// TIA Portal V17 export
// export: Created 2025-03-18T12:31:06.7094667Z, ExportSetting WithDefaults, DisplayName Totally Integrated Automation Portal, DisplayVersion V17 Update 8, DisplayName TIA Portal Openness, DisplayVersion V17 Update 8, DisplayName TIA Portal Version Control Interface, DisplayVersion V17, DisplayName SINAMICS Startdrive Advanced, DisplayVersion V17 SP2, DisplayName SINAMICS Startdrive G110M, G120, G120C, G120D, G120P, G115D, DisplayVersion V17 SP2, DisplayName SINAMICS Startdrive G130, G150, S120, S150, SINAMICS MV, S210, DisplayVersion V17 SP2, DisplayName STEP 7 Professional, DisplayVersion V17 Update 8, DisplayName SINUMERIK ONE STEP 7 Toolbox, DisplayVersion V17 Update 12, DisplayName SINUMERIK 840D sl STEP 7 Toolbox, DisplayVersion V17 Update 12, DisplayName STEP 7 Safety, DisplayVersion V17 Update 6, DisplayName WinCC Advanced, DisplayVersion V17 Update 8
FUNCTION "FC1312_HOME_UNIT_03_STATION_0" : Void   // FC1312, LAD
{ S7_Optimized_Access := 'FALSE' }
AUTHOR : ETXETAR
VERSION : 1.0
// stored: AutoNumber false, IsIECCheckEnabled false, SetENOAutomatically false, UDAEnableTagReadback false
   VAR_TEMP
      UNIT_03_LOCAL_E_RETURNS : Bool;   // UNIT 03 LOCAL E RETURNS
      UNIT_03_MACHINE_E_RETURNS : Bool;   // UNIT 03 MACHINE E RETURNS
   END_VAR
   VAR CONSTANT
      FC_NUMBER : DInt := 1312;
   END_VAR
   VAR_TEMP   // added for the SCL form of the ladder/FBD networks
      _w1 : Bool;
   END_VAR
BEGIN

REGION Network 1: GENERAL CONDITIONS
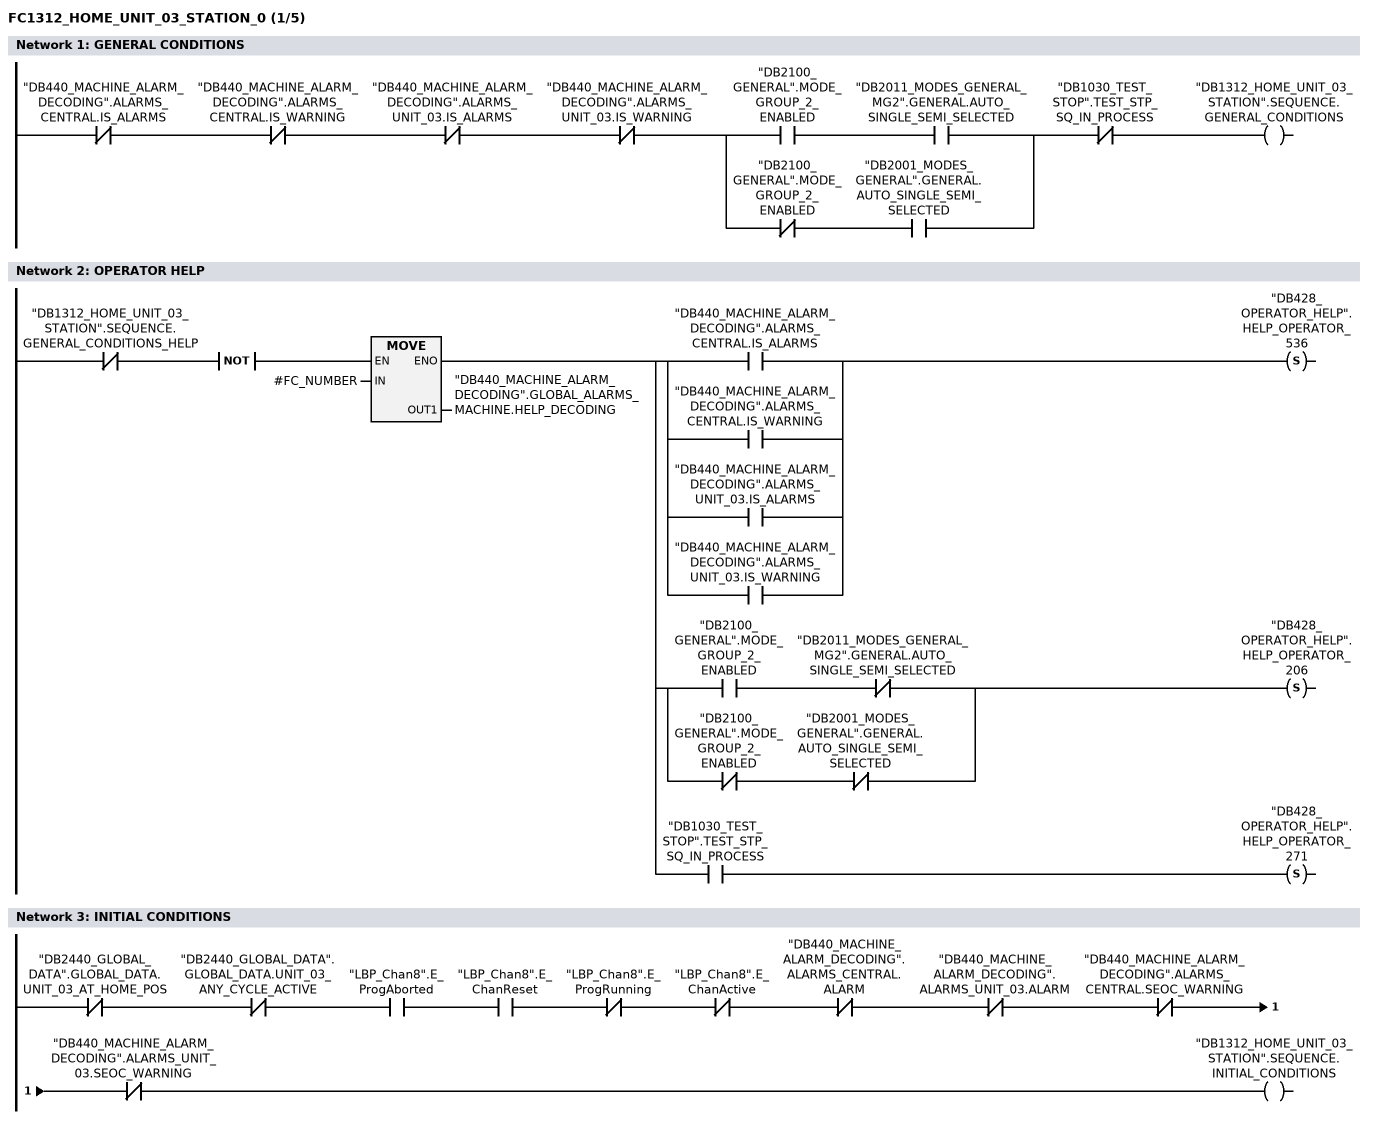
   RUNG wire#powerrail
      I_Contact( "DB440_MACHINE_ALARM_DECODING".ALARMS_CENTRAL.IS_ALARMS )
      I_Contact( "DB440_MACHINE_ALARM_DECODING".ALARMS_CENTRAL.IS_WARNING )
      I_Contact( "DB440_MACHINE_ALARM_DECODING".ALARMS_UNIT_03.IS_ALARMS )
      I_Contact( "DB440_MACHINE_ALARM_DECODING".ALARMS_UNIT_03.IS_WARNING )
      wire#w1
      Contact( "DB2100_GENERAL".MODE_GROUP_2_ENABLED )
      Contact( "DB2011_MODES_GENERAL_MG2".GENERAL.AUTO_SINGLE_SEMI_SELECTED )
      wire#w2
      I_Contact( "DB1030_TEST_STOP".TEST_STP_SQ_IN_PROCESS )
      Coil( "DB1312_HOME_UNIT_03_STATION".SEQUENCE.GENERAL_CONDITIONS )
   END_RUNG
   RUNG wire#w1
      I_Contact( "DB2100_GENERAL".MODE_GROUP_2_ENABLED )
      Contact( "DB2001_MODES_GENERAL".GENERAL.AUTO_SINGLE_SEMI_SELECTED )
   END_RUNG wire#w2
   // the same network as SCL:
   "DB1312_HOME_UNIT_03_STATION".SEQUENCE.GENERAL_CONDITIONS := NOT "DB440_MACHINE_ALARM_DECODING".ALARMS_CENTRAL.IS_ALARMS AND NOT "DB440_MACHINE_ALARM_DECODING".ALARMS_CENTRAL.IS_WARNING AND NOT "DB440_MACHINE_ALARM_DECODING".ALARMS_UNIT_03.IS_ALARMS AND NOT "DB440_MACHINE_ALARM_DECODING".ALARMS_UNIT_03.IS_WARNING AND (("DB2100_GENERAL".MODE_GROUP_2_ENABLED AND "DB2011_MODES_GENERAL_MG2".GENERAL.AUTO_SINGLE_SEMI_SELECTED) OR (NOT "DB2100_GENERAL".MODE_GROUP_2_ENABLED AND "DB2001_MODES_GENERAL".GENERAL.AUTO_SINGLE_SEMI_SELECTED)) AND NOT "DB1030_TEST_STOP".TEST_STP_SQ_IN_PROCESS;
END_REGION

REGION Network 2: OPERATOR HELP
   RUNG wire#powerrail
      I_Contact( "DB1312_HOME_UNIT_03_STATION".SEQUENCE.GENERAL_CONDITIONS_HELP )
      Not()
      { S7_GenerateENO := "TRUE" } Move(in := #FC_NUMBER, out1 => "DB440_MACHINE_ALARM_DECODING".GLOBAL_ALARMS_MACHINE.HELP_DECODING)
      wire#w1
      Contact( "DB440_MACHINE_ALARM_DECODING".ALARMS_CENTRAL.IS_ALARMS )
      wire#w2
      S_Coil( "DB428_OPERATOR_HELP".HELP_OPERATOR_536 )
   END_RUNG
   RUNG wire#w1
      Contact( "DB440_MACHINE_ALARM_DECODING".ALARMS_CENTRAL.IS_WARNING )
   END_RUNG wire#w2
   RUNG wire#w1
      Contact( "DB440_MACHINE_ALARM_DECODING".ALARMS_UNIT_03.IS_ALARMS )
   END_RUNG wire#w2
   RUNG wire#w1
      Contact( "DB440_MACHINE_ALARM_DECODING".ALARMS_UNIT_03.IS_WARNING )
   END_RUNG wire#w2
   RUNG wire#w1
      Contact( "DB2100_GENERAL".MODE_GROUP_2_ENABLED )
      I_Contact( "DB2011_MODES_GENERAL_MG2".GENERAL.AUTO_SINGLE_SEMI_SELECTED )
      wire#w3
      S_Coil( "DB428_OPERATOR_HELP".HELP_OPERATOR_206 )
   END_RUNG
   RUNG wire#w1
      I_Contact( "DB2100_GENERAL".MODE_GROUP_2_ENABLED )
      I_Contact( "DB2001_MODES_GENERAL".GENERAL.AUTO_SINGLE_SEMI_SELECTED )
   END_RUNG wire#w3
   RUNG wire#w1
      Contact( "DB1030_TEST_STOP".TEST_STP_SQ_IN_PROCESS )
      S_Coil( "DB428_OPERATOR_HELP".HELP_OPERATOR_271 )
   END_RUNG
   // the same network as SCL:
   // ENO of a box is taken as its EN; it also drops when the box reports an error
   #_w1 := NOT (NOT "DB1312_HOME_UNIT_03_STATION".SEQUENCE.GENERAL_CONDITIONS_HELP);
   IF #_w1 THEN "DB440_MACHINE_ALARM_DECODING".GLOBAL_ALARMS_MACHINE.HELP_DECODING := #FC_NUMBER; END_IF;
   IF #_w1 AND ("DB440_MACHINE_ALARM_DECODING".ALARMS_CENTRAL.IS_ALARMS OR "DB440_MACHINE_ALARM_DECODING".ALARMS_CENTRAL.IS_WARNING OR "DB440_MACHINE_ALARM_DECODING".ALARMS_UNIT_03.IS_ALARMS OR "DB440_MACHINE_ALARM_DECODING".ALARMS_UNIT_03.IS_WARNING) THEN
       "DB428_OPERATOR_HELP".HELP_OPERATOR_536 := TRUE;
   END_IF;
   IF #_w1 AND (("DB2100_GENERAL".MODE_GROUP_2_ENABLED AND NOT "DB2011_MODES_GENERAL_MG2".GENERAL.AUTO_SINGLE_SEMI_SELECTED) OR (NOT "DB2100_GENERAL".MODE_GROUP_2_ENABLED AND NOT "DB2001_MODES_GENERAL".GENERAL.AUTO_SINGLE_SEMI_SELECTED)) THEN
       "DB428_OPERATOR_HELP".HELP_OPERATOR_206 := TRUE;
   END_IF;
   IF #_w1 AND "DB1030_TEST_STOP".TEST_STP_SQ_IN_PROCESS THEN
       "DB428_OPERATOR_HELP".HELP_OPERATOR_271 := TRUE;
   END_IF;
END_REGION

REGION Network 3: INITIAL CONDITIONS
   RUNG wire#powerrail
      I_Contact( "DB2440_GLOBAL_DATA".GLOBAL_DATA.UNIT_03_AT_HOME_POS )
      I_Contact( "DB2440_GLOBAL_DATA".GLOBAL_DATA.UNIT_03_ANY_CYCLE_ACTIVE )
      Contact( "LBP_Chan8".E_ProgAborted )
      Contact( "LBP_Chan8".E_ChanReset )
      I_Contact( "LBP_Chan8".E_ProgRunning )
      I_Contact( "LBP_Chan8".E_ChanActive )
      I_Contact( "DB440_MACHINE_ALARM_DECODING".ALARMS_CENTRAL.ALARM )
      I_Contact( "DB440_MACHINE_ALARM_DECODING".ALARMS_UNIT_03.ALARM )
      I_Contact( "DB440_MACHINE_ALARM_DECODING".ALARMS_CENTRAL.SEOC_WARNING )
      I_Contact( "DB440_MACHINE_ALARM_DECODING".ALARMS_UNIT_03.SEOC_WARNING )
      Coil( "DB1312_HOME_UNIT_03_STATION".SEQUENCE.INITIAL_CONDITIONS )
   END_RUNG
   // the same network as SCL:
   "DB1312_HOME_UNIT_03_STATION".SEQUENCE.INITIAL_CONDITIONS := NOT "DB2440_GLOBAL_DATA".GLOBAL_DATA.UNIT_03_AT_HOME_POS AND NOT "DB2440_GLOBAL_DATA".GLOBAL_DATA.UNIT_03_ANY_CYCLE_ACTIVE AND "LBP_Chan8".E_ProgAborted AND "LBP_Chan8".E_ChanReset AND NOT "LBP_Chan8".E_ProgRunning AND NOT "LBP_Chan8".E_ChanActive AND NOT "DB440_MACHINE_ALARM_DECODING".ALARMS_CENTRAL.ALARM AND NOT "DB440_MACHINE_ALARM_DECODING".ALARMS_UNIT_03.ALARM AND NOT "DB440_MACHINE_ALARM_DECODING".ALARMS_CENTRAL.SEOC_WARNING AND NOT "DB440_MACHINE_ALARM_DECODING".ALARMS_UNIT_03.SEOC_WARNING;
END_REGION

REGION Network 4: OPERATOR HELP
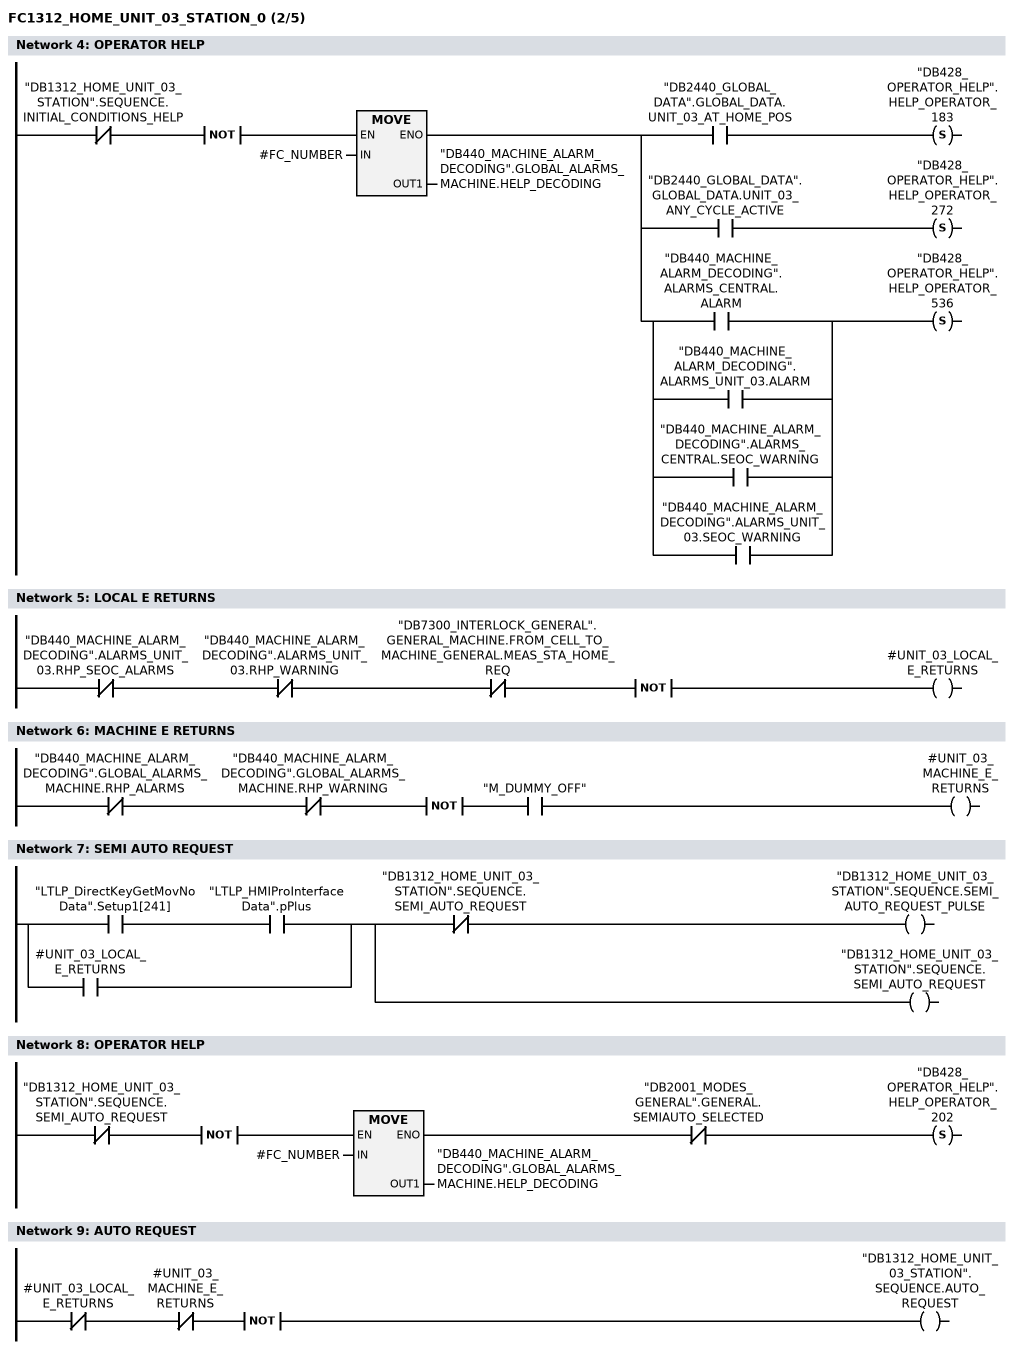
   RUNG wire#powerrail
      I_Contact( "DB1312_HOME_UNIT_03_STATION".SEQUENCE.INITIAL_CONDITIONS_HELP )
      Not()
      { S7_GenerateENO := "TRUE" } Move(in := #FC_NUMBER, out1 => "DB440_MACHINE_ALARM_DECODING".GLOBAL_ALARMS_MACHINE.HELP_DECODING)
      wire#w1
      Contact( "DB2440_GLOBAL_DATA".GLOBAL_DATA.UNIT_03_AT_HOME_POS )
      S_Coil( "DB428_OPERATOR_HELP".HELP_OPERATOR_183 )
   END_RUNG
   RUNG wire#w1
      Contact( "DB2440_GLOBAL_DATA".GLOBAL_DATA.UNIT_03_ANY_CYCLE_ACTIVE )
      S_Coil( "DB428_OPERATOR_HELP".HELP_OPERATOR_272 )
   END_RUNG
   RUNG wire#w1
      Contact( "DB440_MACHINE_ALARM_DECODING".ALARMS_CENTRAL.ALARM )
      wire#w2
      S_Coil( "DB428_OPERATOR_HELP".HELP_OPERATOR_536 )
   END_RUNG
   RUNG wire#w1
      Contact( "DB440_MACHINE_ALARM_DECODING".ALARMS_UNIT_03.ALARM )
   END_RUNG wire#w2
   RUNG wire#w1
      Contact( "DB440_MACHINE_ALARM_DECODING".ALARMS_CENTRAL.SEOC_WARNING )
   END_RUNG wire#w2
   RUNG wire#w1
      Contact( "DB440_MACHINE_ALARM_DECODING".ALARMS_UNIT_03.SEOC_WARNING )
   END_RUNG wire#w2
   // the same network as SCL:
   // ENO of a box is taken as its EN; it also drops when the box reports an error
   #_w1 := NOT (NOT "DB1312_HOME_UNIT_03_STATION".SEQUENCE.INITIAL_CONDITIONS_HELP);
   IF #_w1 THEN "DB440_MACHINE_ALARM_DECODING".GLOBAL_ALARMS_MACHINE.HELP_DECODING := #FC_NUMBER; END_IF;
   IF #_w1 AND "DB2440_GLOBAL_DATA".GLOBAL_DATA.UNIT_03_AT_HOME_POS THEN
       "DB428_OPERATOR_HELP".HELP_OPERATOR_183 := TRUE;
   END_IF;
   IF #_w1 AND "DB2440_GLOBAL_DATA".GLOBAL_DATA.UNIT_03_ANY_CYCLE_ACTIVE THEN
       "DB428_OPERATOR_HELP".HELP_OPERATOR_272 := TRUE;
   END_IF;
   IF #_w1 AND ("DB440_MACHINE_ALARM_DECODING".ALARMS_CENTRAL.ALARM OR "DB440_MACHINE_ALARM_DECODING".ALARMS_UNIT_03.ALARM OR "DB440_MACHINE_ALARM_DECODING".ALARMS_CENTRAL.SEOC_WARNING OR "DB440_MACHINE_ALARM_DECODING".ALARMS_UNIT_03.SEOC_WARNING) THEN
       "DB428_OPERATOR_HELP".HELP_OPERATOR_536 := TRUE;
   END_IF;
END_REGION

REGION Network 5: LOCAL E RETURNS
   RUNG wire#powerrail
      I_Contact( "DB440_MACHINE_ALARM_DECODING".ALARMS_UNIT_03.RHP_SEOC_ALARMS )
      I_Contact( "DB440_MACHINE_ALARM_DECODING".ALARMS_UNIT_03.RHP_WARNING )
      I_Contact( "DB7300_INTERLOCK_GENERAL".GENERAL_MACHINE.FROM_CELL_TO_MACHINE_GENERAL.MEAS_STA_HOME_REQ )
      Not()
      Coil( #UNIT_03_LOCAL_E_RETURNS )
   END_RUNG
   // the same network as SCL:
   #UNIT_03_LOCAL_E_RETURNS := NOT (NOT "DB440_MACHINE_ALARM_DECODING".ALARMS_UNIT_03.RHP_SEOC_ALARMS AND NOT "DB440_MACHINE_ALARM_DECODING".ALARMS_UNIT_03.RHP_WARNING AND NOT "DB7300_INTERLOCK_GENERAL".GENERAL_MACHINE.FROM_CELL_TO_MACHINE_GENERAL.MEAS_STA_HOME_REQ);
END_REGION

REGION Network 6: MACHINE E RETURNS
   RUNG wire#powerrail
      I_Contact( "DB440_MACHINE_ALARM_DECODING".GLOBAL_ALARMS_MACHINE.RHP_ALARMS )
      I_Contact( "DB440_MACHINE_ALARM_DECODING".GLOBAL_ALARMS_MACHINE.RHP_WARNING )
      Not()
      Contact( "M_DUMMY_OFF" )
      Coil( #UNIT_03_MACHINE_E_RETURNS )
   END_RUNG
   // the same network as SCL:
   #UNIT_03_MACHINE_E_RETURNS := NOT (NOT "DB440_MACHINE_ALARM_DECODING".GLOBAL_ALARMS_MACHINE.RHP_ALARMS AND NOT "DB440_MACHINE_ALARM_DECODING".GLOBAL_ALARMS_MACHINE.RHP_WARNING) AND "M_DUMMY_OFF";
END_REGION

REGION Network 7: SEMI AUTO REQUEST
   RUNG wire#powerrail
      Contact( "LTLP_DirectKeyGetMovNoData".Setup1[241] )
      Contact( "LTLP_HMIProInterfaceData".pPlus )
      wire#w1
      I_Contact( "DB1312_HOME_UNIT_03_STATION".SEQUENCE.SEMI_AUTO_REQUEST )
      Coil( "DB1312_HOME_UNIT_03_STATION".SEQUENCE.SEMI_AUTO_REQUEST_PULSE )
   END_RUNG
   RUNG wire#powerrail
      Contact( #UNIT_03_LOCAL_E_RETURNS )
   END_RUNG wire#w1
   RUNG wire#w1
      Coil( "DB1312_HOME_UNIT_03_STATION".SEQUENCE.SEMI_AUTO_REQUEST )
   END_RUNG
   // the same network as SCL:
   #_w1 := ("LTLP_DirectKeyGetMovNoData".Setup1[241] AND "LTLP_HMIProInterfaceData".pPlus) OR #UNIT_03_LOCAL_E_RETURNS;
   "DB1312_HOME_UNIT_03_STATION".SEQUENCE.SEMI_AUTO_REQUEST_PULSE := #_w1 AND NOT "DB1312_HOME_UNIT_03_STATION".SEQUENCE.SEMI_AUTO_REQUEST;
   "DB1312_HOME_UNIT_03_STATION".SEQUENCE.SEMI_AUTO_REQUEST := #_w1;
END_REGION

REGION Network 8: OPERATOR HELP
   RUNG wire#powerrail
      I_Contact( "DB1312_HOME_UNIT_03_STATION".SEQUENCE.SEMI_AUTO_REQUEST )
      Not()
      { S7_GenerateENO := "TRUE" } Move(in := #FC_NUMBER, out1 => "DB440_MACHINE_ALARM_DECODING".GLOBAL_ALARMS_MACHINE.HELP_DECODING)
      I_Contact( "DB2001_MODES_GENERAL".GENERAL.SEMIAUTO_SELECTED )
      S_Coil( "DB428_OPERATOR_HELP".HELP_OPERATOR_202 )
   END_RUNG
   // the same network as SCL:
   // ENO of a box is taken as its EN; it also drops when the box reports an error
   #_w1 := NOT (NOT "DB1312_HOME_UNIT_03_STATION".SEQUENCE.SEMI_AUTO_REQUEST);
   IF #_w1 THEN "DB440_MACHINE_ALARM_DECODING".GLOBAL_ALARMS_MACHINE.HELP_DECODING := #FC_NUMBER; END_IF;
   IF #_w1 AND NOT "DB2001_MODES_GENERAL".GENERAL.SEMIAUTO_SELECTED THEN
       "DB428_OPERATOR_HELP".HELP_OPERATOR_202 := TRUE;
   END_IF;
END_REGION

REGION Network 9: AUTO REQUEST
   RUNG wire#powerrail
      I_Contact( #UNIT_03_LOCAL_E_RETURNS )
      I_Contact( #UNIT_03_MACHINE_E_RETURNS )
      Not()
      Coil( "DB1312_HOME_UNIT_03_STATION".SEQUENCE.AUTO_REQUEST )
   END_RUNG
   // the same network as SCL:
   "DB1312_HOME_UNIT_03_STATION".SEQUENCE.AUTO_REQUEST := NOT (NOT #UNIT_03_LOCAL_E_RETURNS AND NOT #UNIT_03_MACHINE_E_RETURNS);
END_REGION

REGION Network 10: REQUEST
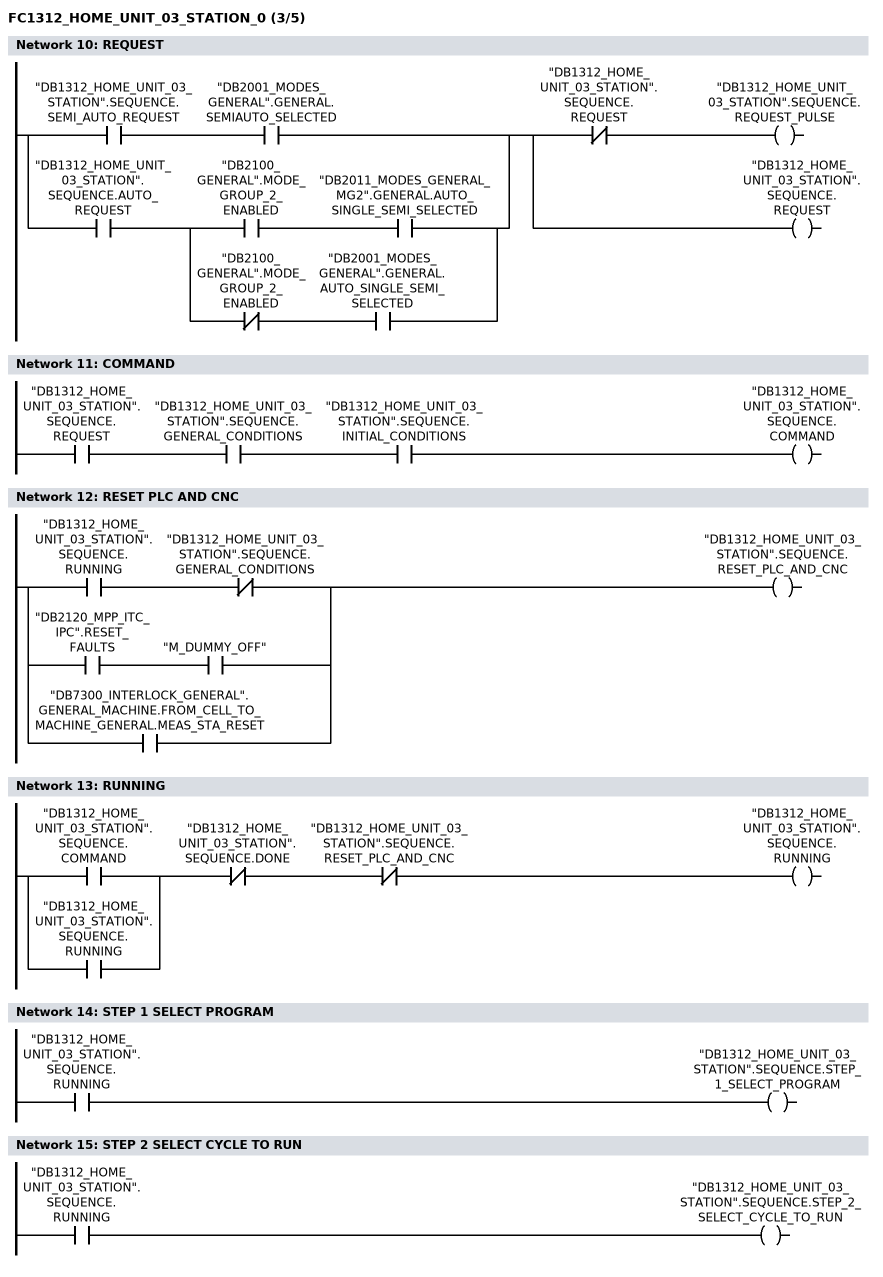
   RUNG wire#powerrail
      Contact( "DB1312_HOME_UNIT_03_STATION".SEQUENCE.SEMI_AUTO_REQUEST )
      Contact( "DB2001_MODES_GENERAL".GENERAL.SEMIAUTO_SELECTED )
      wire#w1
      I_Contact( "DB1312_HOME_UNIT_03_STATION".SEQUENCE.REQUEST )
      Coil( "DB1312_HOME_UNIT_03_STATION".SEQUENCE.REQUEST_PULSE )
   END_RUNG
   RUNG wire#powerrail
      Contact( "DB1312_HOME_UNIT_03_STATION".SEQUENCE.AUTO_REQUEST )
      wire#w2
      Contact( "DB2100_GENERAL".MODE_GROUP_2_ENABLED )
      Contact( "DB2011_MODES_GENERAL_MG2".GENERAL.AUTO_SINGLE_SEMI_SELECTED )
   END_RUNG wire#w1
   RUNG wire#w2
      I_Contact( "DB2100_GENERAL".MODE_GROUP_2_ENABLED )
      Contact( "DB2001_MODES_GENERAL".GENERAL.AUTO_SINGLE_SEMI_SELECTED )
   END_RUNG wire#w1
   RUNG wire#w1
      Coil( "DB1312_HOME_UNIT_03_STATION".SEQUENCE.REQUEST )
   END_RUNG
   // the same network as SCL:
   #_w1 := ("DB1312_HOME_UNIT_03_STATION".SEQUENCE.SEMI_AUTO_REQUEST AND "DB2001_MODES_GENERAL".GENERAL.SEMIAUTO_SELECTED) OR ("DB1312_HOME_UNIT_03_STATION".SEQUENCE.AUTO_REQUEST AND (("DB2100_GENERAL".MODE_GROUP_2_ENABLED AND "DB2011_MODES_GENERAL_MG2".GENERAL.AUTO_SINGLE_SEMI_SELECTED) OR (NOT "DB2100_GENERAL".MODE_GROUP_2_ENABLED AND "DB2001_MODES_GENERAL".GENERAL.AUTO_SINGLE_SEMI_SELECTED)));
   "DB1312_HOME_UNIT_03_STATION".SEQUENCE.REQUEST_PULSE := #_w1 AND NOT "DB1312_HOME_UNIT_03_STATION".SEQUENCE.REQUEST;
   "DB1312_HOME_UNIT_03_STATION".SEQUENCE.REQUEST := #_w1;
END_REGION

REGION Network 11: COMMAND
   RUNG wire#powerrail
      Contact( "DB1312_HOME_UNIT_03_STATION".SEQUENCE.REQUEST )
      Contact( "DB1312_HOME_UNIT_03_STATION".SEQUENCE.GENERAL_CONDITIONS )
      Contact( "DB1312_HOME_UNIT_03_STATION".SEQUENCE.INITIAL_CONDITIONS )
      Coil( "DB1312_HOME_UNIT_03_STATION".SEQUENCE.COMMAND )
   END_RUNG
   // the same network as SCL:
   "DB1312_HOME_UNIT_03_STATION".SEQUENCE.COMMAND := "DB1312_HOME_UNIT_03_STATION".SEQUENCE.REQUEST AND "DB1312_HOME_UNIT_03_STATION".SEQUENCE.GENERAL_CONDITIONS AND "DB1312_HOME_UNIT_03_STATION".SEQUENCE.INITIAL_CONDITIONS;
END_REGION

REGION Network 12: RESET PLC AND CNC
   RUNG wire#powerrail
      Contact( "DB1312_HOME_UNIT_03_STATION".SEQUENCE.RUNNING )
      I_Contact( "DB1312_HOME_UNIT_03_STATION".SEQUENCE.GENERAL_CONDITIONS )
      wire#w1
      Coil( "DB1312_HOME_UNIT_03_STATION".SEQUENCE.RESET_PLC_AND_CNC )
   END_RUNG
   RUNG wire#powerrail
      Contact( "DB2120_MPP_ITC_IPC".RESET_FAULTS )
      Contact( "M_DUMMY_OFF" )
   END_RUNG wire#w1
   RUNG wire#powerrail
      Contact( "DB7300_INTERLOCK_GENERAL".GENERAL_MACHINE.FROM_CELL_TO_MACHINE_GENERAL.MEAS_STA_RESET )
   END_RUNG wire#w1
   // the same network as SCL:
   "DB1312_HOME_UNIT_03_STATION".SEQUENCE.RESET_PLC_AND_CNC := ("DB1312_HOME_UNIT_03_STATION".SEQUENCE.RUNNING AND NOT "DB1312_HOME_UNIT_03_STATION".SEQUENCE.GENERAL_CONDITIONS) OR ("DB2120_MPP_ITC_IPC".RESET_FAULTS AND "M_DUMMY_OFF") OR "DB7300_INTERLOCK_GENERAL".GENERAL_MACHINE.FROM_CELL_TO_MACHINE_GENERAL.MEAS_STA_RESET;
END_REGION

REGION Network 13: RUNNING
   RUNG wire#powerrail
      Contact( "DB1312_HOME_UNIT_03_STATION".SEQUENCE.COMMAND )
      wire#w1
      I_Contact( "DB1312_HOME_UNIT_03_STATION".SEQUENCE.DONE )
      I_Contact( "DB1312_HOME_UNIT_03_STATION".SEQUENCE.RESET_PLC_AND_CNC )
      Coil( "DB1312_HOME_UNIT_03_STATION".SEQUENCE.RUNNING )
   END_RUNG
   RUNG wire#powerrail
      Contact( "DB1312_HOME_UNIT_03_STATION".SEQUENCE.RUNNING )
   END_RUNG wire#w1
   // the same network as SCL:
   "DB1312_HOME_UNIT_03_STATION".SEQUENCE.RUNNING := ("DB1312_HOME_UNIT_03_STATION".SEQUENCE.COMMAND OR "DB1312_HOME_UNIT_03_STATION".SEQUENCE.RUNNING) AND NOT "DB1312_HOME_UNIT_03_STATION".SEQUENCE.DONE AND NOT "DB1312_HOME_UNIT_03_STATION".SEQUENCE.RESET_PLC_AND_CNC;
END_REGION

REGION Network 14: STEP 1 SELECT PROGRAM
   RUNG wire#powerrail
      Contact( "DB1312_HOME_UNIT_03_STATION".SEQUENCE.RUNNING )
      Coil( "DB1312_HOME_UNIT_03_STATION".SEQUENCE.STEP_1_SELECT_PROGRAM )
   END_RUNG
   // the same network as SCL:
   "DB1312_HOME_UNIT_03_STATION".SEQUENCE.STEP_1_SELECT_PROGRAM := "DB1312_HOME_UNIT_03_STATION".SEQUENCE.RUNNING;
END_REGION

REGION Network 15: STEP 2 SELECT CYCLE TO RUN
   RUNG wire#powerrail
      Contact( "DB1312_HOME_UNIT_03_STATION".SEQUENCE.RUNNING )
      Coil( "DB1312_HOME_UNIT_03_STATION".SEQUENCE.STEP_2_SELECT_CYCLE_TO_RUN )
   END_RUNG
   // the same network as SCL:
   "DB1312_HOME_UNIT_03_STATION".SEQUENCE.STEP_2_SELECT_CYCLE_TO_RUN := "DB1312_HOME_UNIT_03_STATION".SEQUENCE.RUNNING;
END_REGION

REGION Network 16: STEP 3 RUN CNC PROGRAM
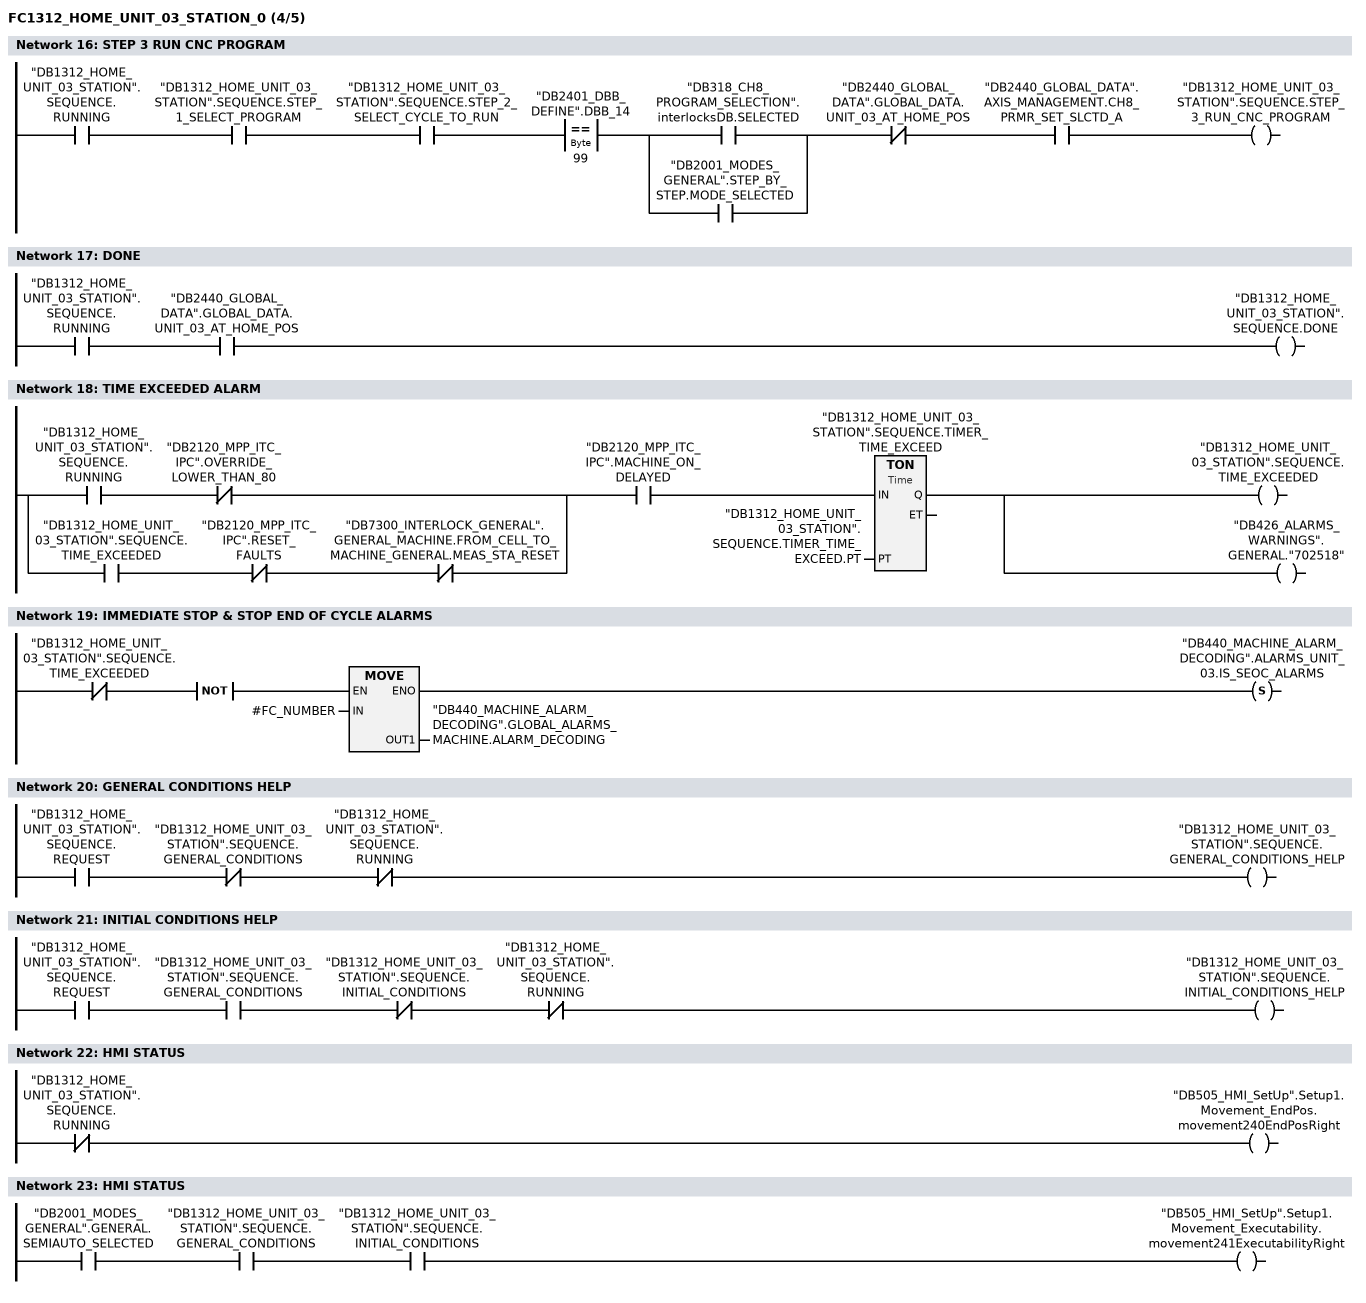
   RUNG wire#powerrail
      Contact( "DB1312_HOME_UNIT_03_STATION".SEQUENCE.RUNNING )
      Contact( "DB1312_HOME_UNIT_03_STATION".SEQUENCE.STEP_1_SELECT_PROGRAM )
      Contact( "DB1312_HOME_UNIT_03_STATION".SEQUENCE.STEP_2_SELECT_CYCLE_TO_RUN )
      { S7_Templates := "SrcType := Byte" } EQ_Contact(in1 := "DB2401_DBB_DEFINE".DBB_14, in2 := 99)
      wire#w1
      Contact( "DB318_CH8_PROGRAM_SELECTION".interlocksDB.SELECTED )
      wire#w2
      I_Contact( "DB2440_GLOBAL_DATA".GLOBAL_DATA.UNIT_03_AT_HOME_POS )
      Contact( "DB2440_GLOBAL_DATA".AXIS_MANAGEMENT.CH8_PRMR_SET_SLCTD_A )
      Coil( "DB1312_HOME_UNIT_03_STATION".SEQUENCE.STEP_3_RUN_CNC_PROGRAM )
   END_RUNG
   RUNG wire#w1
      Contact( "DB2001_MODES_GENERAL".STEP_BY_STEP.MODE_SELECTED )
   END_RUNG wire#w2
   // the same network as SCL:
   "DB1312_HOME_UNIT_03_STATION".SEQUENCE.STEP_3_RUN_CNC_PROGRAM := "DB1312_HOME_UNIT_03_STATION".SEQUENCE.RUNNING AND "DB1312_HOME_UNIT_03_STATION".SEQUENCE.STEP_1_SELECT_PROGRAM AND "DB1312_HOME_UNIT_03_STATION".SEQUENCE.STEP_2_SELECT_CYCLE_TO_RUN AND ("DB2401_DBB_DEFINE".DBB_14 = 99) AND ("DB318_CH8_PROGRAM_SELECTION".interlocksDB.SELECTED OR "DB2001_MODES_GENERAL".STEP_BY_STEP.MODE_SELECTED) AND NOT "DB2440_GLOBAL_DATA".GLOBAL_DATA.UNIT_03_AT_HOME_POS AND "DB2440_GLOBAL_DATA".AXIS_MANAGEMENT.CH8_PRMR_SET_SLCTD_A;
END_REGION

REGION Network 17: DONE
   RUNG wire#powerrail
      Contact( "DB1312_HOME_UNIT_03_STATION".SEQUENCE.RUNNING )
      Contact( "DB2440_GLOBAL_DATA".GLOBAL_DATA.UNIT_03_AT_HOME_POS )
      Coil( "DB1312_HOME_UNIT_03_STATION".SEQUENCE.DONE )
   END_RUNG
   // the same network as SCL:
   "DB1312_HOME_UNIT_03_STATION".SEQUENCE.DONE := "DB1312_HOME_UNIT_03_STATION".SEQUENCE.RUNNING AND "DB2440_GLOBAL_DATA".GLOBAL_DATA.UNIT_03_AT_HOME_POS;
END_REGION

REGION Network 18: TIME EXCEEDED ALARM
   RUNG wire#powerrail
      Contact( "DB1312_HOME_UNIT_03_STATION".SEQUENCE.RUNNING )
      I_Contact( "DB2120_MPP_ITC_IPC".OVERRIDE_LOWER_THAN_80 )
      wire#w1
      Contact( "DB2120_MPP_ITC_IPC".MACHINE_ON_DELAYED )
      { S7_Templates := "time_type := Time" } "DB1312_HOME_UNIT_03_STATION".SEQUENCE.TIMER_TIME_EXCEED.TON(pt := "DB1312_HOME_UNIT_03_STATION".SEQUENCE.TIMER_TIME_EXCEED.PT, et =>)
      wire#w2
      Coil( "DB1312_HOME_UNIT_03_STATION".SEQUENCE.TIME_EXCEEDED )
   END_RUNG
   RUNG wire#powerrail
      Contact( "DB1312_HOME_UNIT_03_STATION".SEQUENCE.TIME_EXCEEDED )
      I_Contact( "DB2120_MPP_ITC_IPC".RESET_FAULTS )
      I_Contact( "DB7300_INTERLOCK_GENERAL".GENERAL_MACHINE.FROM_CELL_TO_MACHINE_GENERAL.MEAS_STA_RESET )
   END_RUNG wire#w1
   RUNG wire#w2
      Coil( "DB426_ALARMS_WARNINGS".GENERAL."702518" )
   END_RUNG
   // the same network as SCL:
   "DB1312_HOME_UNIT_03_STATION".SEQUENCE.TIMER_TIME_EXCEED.TON(IN := (("DB1312_HOME_UNIT_03_STATION".SEQUENCE.RUNNING AND NOT "DB2120_MPP_ITC_IPC".OVERRIDE_LOWER_THAN_80) OR ("DB1312_HOME_UNIT_03_STATION".SEQUENCE.TIME_EXCEEDED AND NOT "DB2120_MPP_ITC_IPC".RESET_FAULTS AND NOT "DB7300_INTERLOCK_GENERAL".GENERAL_MACHINE.FROM_CELL_TO_MACHINE_GENERAL.MEAS_STA_RESET)) AND "DB2120_MPP_ITC_IPC".MACHINE_ON_DELAYED,
                           PT := "DB1312_HOME_UNIT_03_STATION".SEQUENCE.TIMER_TIME_EXCEED.PT);
   "DB1312_HOME_UNIT_03_STATION".SEQUENCE.TIME_EXCEEDED := "DB1312_HOME_UNIT_03_STATION".SEQUENCE.TIMER_TIME_EXCEED.Q;
   "DB426_ALARMS_WARNINGS".GENERAL."702518" := "DB1312_HOME_UNIT_03_STATION".SEQUENCE.TIMER_TIME_EXCEED.Q;
END_REGION

REGION Network 19: IMMEDIATE STOP & STOP END OF CYCLE ALARMS
   RUNG wire#powerrail
      I_Contact( "DB1312_HOME_UNIT_03_STATION".SEQUENCE.TIME_EXCEEDED )
      Not()
      { S7_GenerateENO := "TRUE" } Move(in := #FC_NUMBER, out1 => "DB440_MACHINE_ALARM_DECODING".GLOBAL_ALARMS_MACHINE.ALARM_DECODING)
      S_Coil( "DB440_MACHINE_ALARM_DECODING".ALARMS_UNIT_03.IS_SEOC_ALARMS )
   END_RUNG
   // the same network as SCL:
   // ENO of a box is taken as its EN; it also drops when the box reports an error
   IF NOT (NOT "DB1312_HOME_UNIT_03_STATION".SEQUENCE.TIME_EXCEEDED) THEN
       "DB440_MACHINE_ALARM_DECODING".GLOBAL_ALARMS_MACHINE.ALARM_DECODING := #FC_NUMBER;
       "DB440_MACHINE_ALARM_DECODING".ALARMS_UNIT_03.IS_SEOC_ALARMS := TRUE;
   END_IF;
END_REGION

REGION Network 20: GENERAL CONDITIONS HELP
   RUNG wire#powerrail
      Contact( "DB1312_HOME_UNIT_03_STATION".SEQUENCE.REQUEST )
      I_Contact( "DB1312_HOME_UNIT_03_STATION".SEQUENCE.GENERAL_CONDITIONS )
      I_Contact( "DB1312_HOME_UNIT_03_STATION".SEQUENCE.RUNNING )
      Coil( "DB1312_HOME_UNIT_03_STATION".SEQUENCE.GENERAL_CONDITIONS_HELP )
   END_RUNG
   // the same network as SCL:
   "DB1312_HOME_UNIT_03_STATION".SEQUENCE.GENERAL_CONDITIONS_HELP := "DB1312_HOME_UNIT_03_STATION".SEQUENCE.REQUEST AND NOT "DB1312_HOME_UNIT_03_STATION".SEQUENCE.GENERAL_CONDITIONS AND NOT "DB1312_HOME_UNIT_03_STATION".SEQUENCE.RUNNING;
END_REGION

REGION Network 21: INITIAL CONDITIONS HELP
   RUNG wire#powerrail
      Contact( "DB1312_HOME_UNIT_03_STATION".SEQUENCE.REQUEST )
      Contact( "DB1312_HOME_UNIT_03_STATION".SEQUENCE.GENERAL_CONDITIONS )
      I_Contact( "DB1312_HOME_UNIT_03_STATION".SEQUENCE.INITIAL_CONDITIONS )
      I_Contact( "DB1312_HOME_UNIT_03_STATION".SEQUENCE.RUNNING )
      Coil( "DB1312_HOME_UNIT_03_STATION".SEQUENCE.INITIAL_CONDITIONS_HELP )
   END_RUNG
   // the same network as SCL:
   "DB1312_HOME_UNIT_03_STATION".SEQUENCE.INITIAL_CONDITIONS_HELP := "DB1312_HOME_UNIT_03_STATION".SEQUENCE.REQUEST AND "DB1312_HOME_UNIT_03_STATION".SEQUENCE.GENERAL_CONDITIONS AND NOT "DB1312_HOME_UNIT_03_STATION".SEQUENCE.INITIAL_CONDITIONS AND NOT "DB1312_HOME_UNIT_03_STATION".SEQUENCE.RUNNING;
END_REGION

REGION Network 22: HMI STATUS
   RUNG wire#powerrail
      I_Contact( "DB1312_HOME_UNIT_03_STATION".SEQUENCE.RUNNING )
      Coil( "DB505_HMI_SetUp".Setup1.Movement_EndPos.movement240EndPosRight )
   END_RUNG
   // the same network as SCL:
   "DB505_HMI_SetUp".Setup1.Movement_EndPos.movement240EndPosRight := NOT "DB1312_HOME_UNIT_03_STATION".SEQUENCE.RUNNING;
END_REGION

REGION Network 23: HMI STATUS
   RUNG wire#powerrail
      Contact( "DB2001_MODES_GENERAL".GENERAL.SEMIAUTO_SELECTED )
      Contact( "DB1312_HOME_UNIT_03_STATION".SEQUENCE.GENERAL_CONDITIONS )
      Contact( "DB1312_HOME_UNIT_03_STATION".SEQUENCE.INITIAL_CONDITIONS )
      Coil( "DB505_HMI_SetUp".Setup1.Movement_Executability.movement241ExecutabilityRight )
   END_RUNG
   // the same network as SCL:
   "DB505_HMI_SetUp".Setup1.Movement_Executability.movement241ExecutabilityRight := "DB2001_MODES_GENERAL".GENERAL.SEMIAUTO_SELECTED AND "DB1312_HOME_UNIT_03_STATION".SEQUENCE.GENERAL_CONDITIONS AND "DB1312_HOME_UNIT_03_STATION".SEQUENCE.INITIAL_CONDITIONS;
END_REGION

REGION Network 24: HMI STATUS
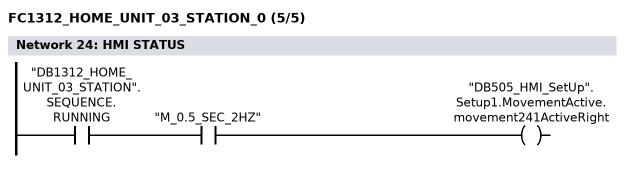
   RUNG wire#powerrail
      Contact( "DB1312_HOME_UNIT_03_STATION".SEQUENCE.RUNNING )
      Contact( "M_0.5_SEC_2HZ" )
      Coil( "DB505_HMI_SetUp".Setup1.MovementActive.movement241ActiveRight )
   END_RUNG
   // the same network as SCL:
   "DB505_HMI_SetUp".Setup1.MovementActive.movement241ActiveRight := "DB1312_HOME_UNIT_03_STATION".SEQUENCE.RUNNING AND "M_0.5_SEC_2HZ";
END_REGION
END_FUNCTION
